(* Logix 5000 project; controller Corte_Silla vendor 1 type 14 code 156 rev 30.11; software revision 30.00 *)

TASK MainTask (continuous, watchdog 500 ms) : MainProgram

MODULES
   Local : vendor 1 type 14 code 156 (Compact 0, rev 30.11)
END_MODULES

PROGRAM MainProgram   (* main routine Memorizacion_de_etapas *)
VAR
   A1 : BOOL;   // Banda 1
   A2 : BOOL;   // Banda 2
   A3 : BOOL;   // Gripper
   Cont1 : COUNTER := (PRE := 12);
   Cont2 : COUNTER := (PRE := 12);
   Cont3 : COUNTER;
   Cont4 : COUNTER;
   Cont5 : COUNTER;
   Cont6 : COUNTER;
   DI_01 : BOOL;
   DI_02 : BOOL;
   DI_03 : BOOL;
   DI_04 : BOOL;
   DI_05 : BOOL;
   DI_06 : BOOL;
   DI_07 : BOOL;
   DI_08 : BOOL;
   DI_09 : BOOL;
   DI_10 : BOOL;
   DO_01 : BOOL;
   DO_02 : BOOL;
   DO_03 : BOOL;
   DO_04 : BOOL;
   DO_05 : BOOL;
   DO_06 : BOOL;
   DO_07 : BOOL;
   DO_08 : BOOL;
   DO_09 : BOOL;
   DO_10 : BOOL;
   Dobladora_DN : BOOL;
   E0 : BOOL;
   E1 : BOOL;
   E10 : BOOL;
   E11 : BOOL;
   E12 : BOOL;
   E13 : BOOL;
   E14 : BOOL;
   E15 : BOOL;
   E16 : BOOL;
   E17 : BOOL;
   E18 : BOOL;
   E19 : BOOL;
   E2 : BOOL;
   E20 : BOOL;
   E21 : BOOL;
   E22 : BOOL;
   E3 : BOOL;
   E4 : BOOL;
   E5 : BOOL;
   E6 : BOOL;
   E7 : BOOL;
   E8 : BOOL;
   E9 : BOOL;
   March : BOOL;
   S1 : BOOL;   // Sensor Banda
   S2 : BOOL;   // Sensor_Dobladora
   Start : BOOL;
   Stop : BOOL;
   T01 : TIMER := (PRE := 100);
   T02 : TIMER := (PRE := 1000);
END_VAR

ROUTINE Activacion_de_salidas   (* ladder *)
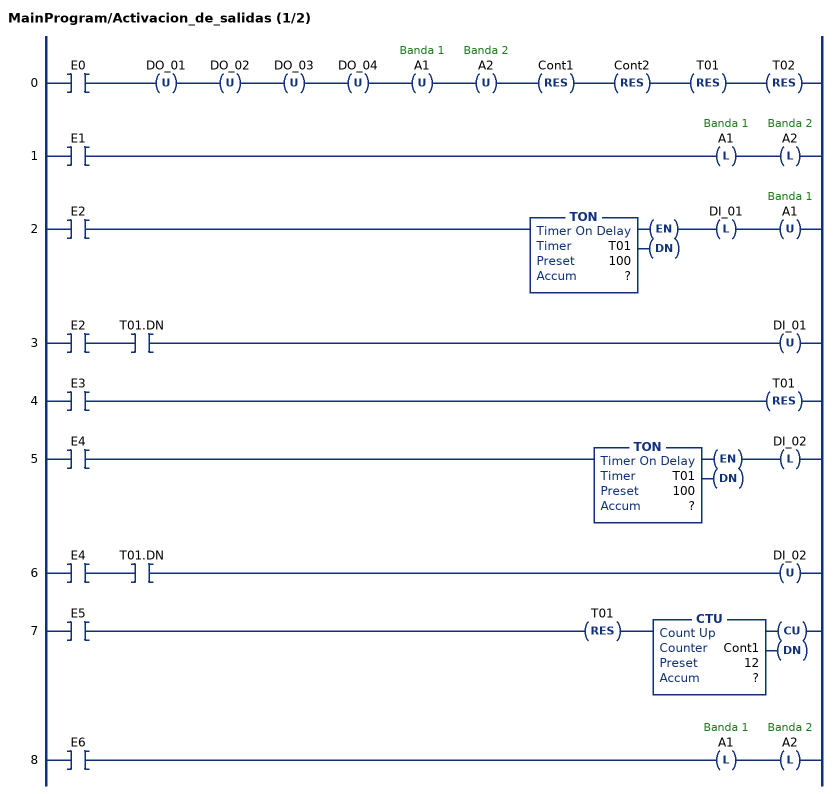
   0: XIC(E0)OTU(DO_01)OTU(DO_02)OTU(DO_03)OTU(DO_04)OTU(A1)OTU(A2)RES(Cont1)RES(Cont2)RES(T01)RES(T02);
   1: XIC(E1)OTL(A1)OTL(A2);
   2: XIC(E2)TON(T01,?,?)OTL(DI_01)OTU(A1);
   3: XIC(E2)XIC(T01.DN)OTU(DI_01);
   4: XIC(E3)RES(T01);
   5: XIC(E4)TON(T01,?,?)OTL(DI_02);
   6: XIC(E4)XIC(T01.DN)OTU(DI_02);
   7: XIC(E5)RES(T01)CTU(Cont1,?,?);
   8: XIC(E6)OTL(A1)OTL(A2);
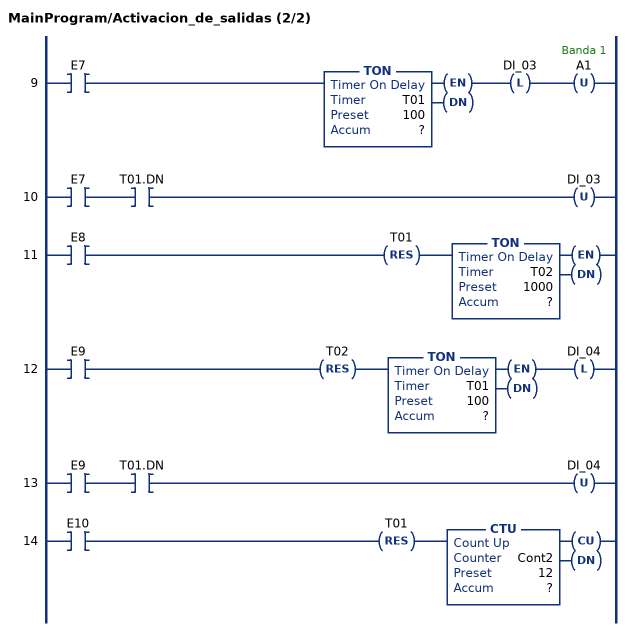
   9: XIC(E7)TON(T01,?,?)OTL(DI_03)OTU(A1);
   10: XIC(E7)XIC(T01.DN)OTU(DI_03);
   11: XIC(E8)RES(T01)TON(T02,?,?);
   12: XIC(E9)RES(T02)TON(T01,?,?)OTL(DI_04);
   13: XIC(E9)XIC(T01.DN)OTU(DI_04);
   14: XIC(E10)RES(T01)CTU(Cont2,?,?);
END_ROUTINE

ROUTINE Memorizacion_de_etapas   (* ladder *)
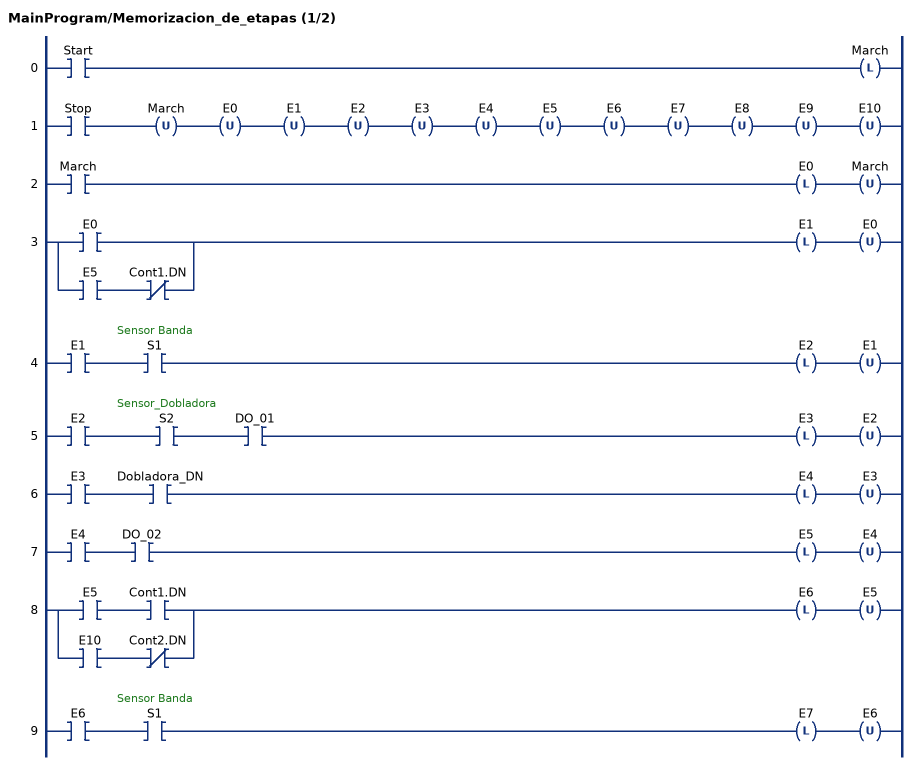
   0: XIC(Start)OTL(March);
   1: XIC(Stop)OTU(March)OTU(E0)OTU(E1)OTU(E2)OTU(E3)OTU(E4)OTU(E5)OTU(E6)OTU(E7)OTU(E8)OTU(E9)OTU(E10);
   2: XIC(March)OTL(E0)OTU(March);
   3: [XIC(E0) ,XIC(E5) XIO(Cont1.DN) ]OTL(E1)OTU(E0);
   4: XIC(E1)XIC(S1)OTL(E2)OTU(E1);
   5: XIC(E2)XIC(S2)XIC(DO_01)OTL(E3)OTU(E2);
   6: XIC(E3)XIC(Dobladora_DN)OTL(E4)OTU(E3);
   7: XIC(E4)XIC(DO_02)OTL(E5)OTU(E4);
   8: [XIC(E5) XIC(Cont1.DN) ,XIC(E10) XIO(Cont2.DN) ]OTL(E6)OTU(E5);
   9: XIC(E6)XIC(S1)OTL(E7)OTU(E6);
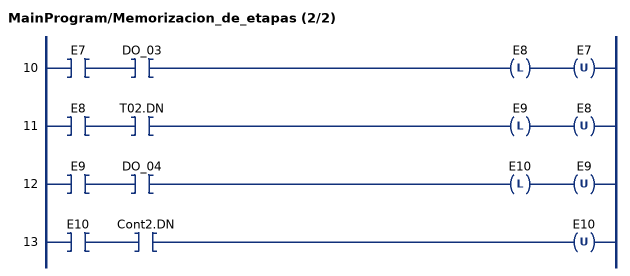
   10: XIC(E7)XIC(DO_03)OTL(E8)OTU(E7);
   11: XIC(E8)XIC(T02.DN)OTL(E9)OTU(E8);
   12: XIC(E9)XIC(DO_04)OTL(E10)OTU(E9);
   13: XIC(E10)XIC(Cont2.DN)OTU(E10);
END_ROUTINE
END_PROGRAM
